{attribute 'GeneratedUsingTerminal: EK1122-0000-0018'}
{attribute addProperty BoxType "EK1122-0000-0018"}
{attribute addProperty Id "Beckhoff_EL33xxsub_EK1100EK1100_1FC0878B2"}
{attribute addProperty CRC "4081559662"}
{attribute addProperty Size "2"}
TYPE Beckhoff_EL33xxEK1122_F347A86E EXTENDS EK1122_1FC0878B :
STRUCT
	{attribute addProperty Name "Beckhoff_EL33xxsub_EK1100"}
	{attribute addProperty PreviousPort "Beckhoff EL33xxEK1122 : D"}
	Beckhoff_EL33xxsub_EK1100 : EK1100_1FC0878B;
END_STRUCT
END_TYPE

(* stored: Version 1.2.0.0, ProductVersion 3.1.4024.9
   DUT Beckhoff_EL33xxEK1122_F347A86E: Id {e96b7982-c292-4d83-bc0b-8756b52114e7} *)
